FUNCTION_BLOCK EL1088
VAR
	_io : EL1xx8_Data;
	{attribute addProperty Name "WcState"}
	_wcState : WcStateInputToggle;
	{attribute addProperty Name "Info data"}
	_infoData : InfoDataBase;
END_VAR

PROPERTY IO : REFERENCE TO EL1xx8_Data
GET
IO REF= _io;
END_GET
END_PROPERTY

PROPERTY WcState : REFERENCE TO WcStateInputToggle
GET
WcState REF= _wcState;
END_GET
END_PROPERTY

END_FUNCTION_BLOCK

(* stored: Version 1.1.0.1, ProductVersion 3.1.4024.9
   POU EL1088: Id {851a3218-8e37-0cc7-3e8c-5cfb2b1cc8fc}, SpecialFunc None
   Property IO: Id {fdd36e46-cf10-092c-360a-5e703a6946c6}
   Get Get: Id {d755e0e0-9818-0f15-01f0-f07d255849f2}
   Property WcState: Id {a317a434-59c5-075c-2db2-6ae762c55d4b}
   Get Get: Id {eb4a8fdc-ccc1-0559-153d-c517c26ea53f} *)
